TYPE st_Powercontrol_PIDparams :
STRUCT
	enable					: BOOL;
	Kp						: REAL;
	Tv						: UINT; //ms
	Tn						: UINT; //ms
	Td						: UINT; //ms
	Outerwindow				: REAL;
	InnerWindow				: REAL;
	OutputDeadband			: REAL;
	InputDeadband			: REAL;
END_STRUCT
END_TYPE

(* stored: Version 1.1.0.1, ProductVersion 3.1.4026.18
   DUT st_Powercontrol_PIDparams: Id {249b63ce-e3fd-47f8-9b6c-d7fb2b8de182} *)
